{attribute addProperty BoxType "EK1100-0000-0018"}
{attribute addProperty Id "Beckhoff_ER2xxxEK1122Beckhoff_ER2xxxEK1122_C26931CF6706838.25"}
{attribute addProperty CRC "3268246309"}
{attribute addProperty SizeInBites "6706"}
{attribute addProperty SizeInBytes "838.25"}
TYPE Beckhoff_ER2xxx_C2CD7B25 EXTENDS EK1100_179A0949 :
STRUCT
	{attribute addProperty Name "Beckhoff_ER2xxxEK1122"}
	Beckhoff_ER2xxxEK1122 : Beckhoff_ER2xxxEK1122_C26931CF;
END_STRUCT
END_TYPE

(* stored: Version 1.2.0.0, ProductVersion 3.1.4024.9
   DUT Beckhoff_ER2xxx_C2CD7B25: Id {5e63ba61-2724-4092-a5e1-b6537cd7a24b} *)
